FUNCTION pv_float_to_dac : INT
VAR_INPUT
	pv			: LREAL;
	pv_max		: LREAL;
	pv_min		: LREAL;
	dac_max		: LREAL;
	dac_min		: LREAL;
END_VAR
VAR
	pv_float_to_dac_old: INT := 0;
END_VAR

IF floatisnan(pv) THEN
	pv_float_to_dac := 0;
ELSE

	IF pv > pv_max THEN
		pv := pv_max;
	END_IF
	IF pv < pv_min THEN
		pv := pv_min;
	END_IF
	pv_float_to_dac := LREAL_TO_INT(  (((dac_max-dac_min)/(pv_max-pv_min))*pv) + dac_min  );

END_IF

END_FUNCTION

(* stored: Version 1.1.0.1, ProductVersion 3.1.0.36
   POU pv_float_to_dac: Id {27287405-a677-4f65-93c1-109ed01550ed}, SpecialFunc None *)
